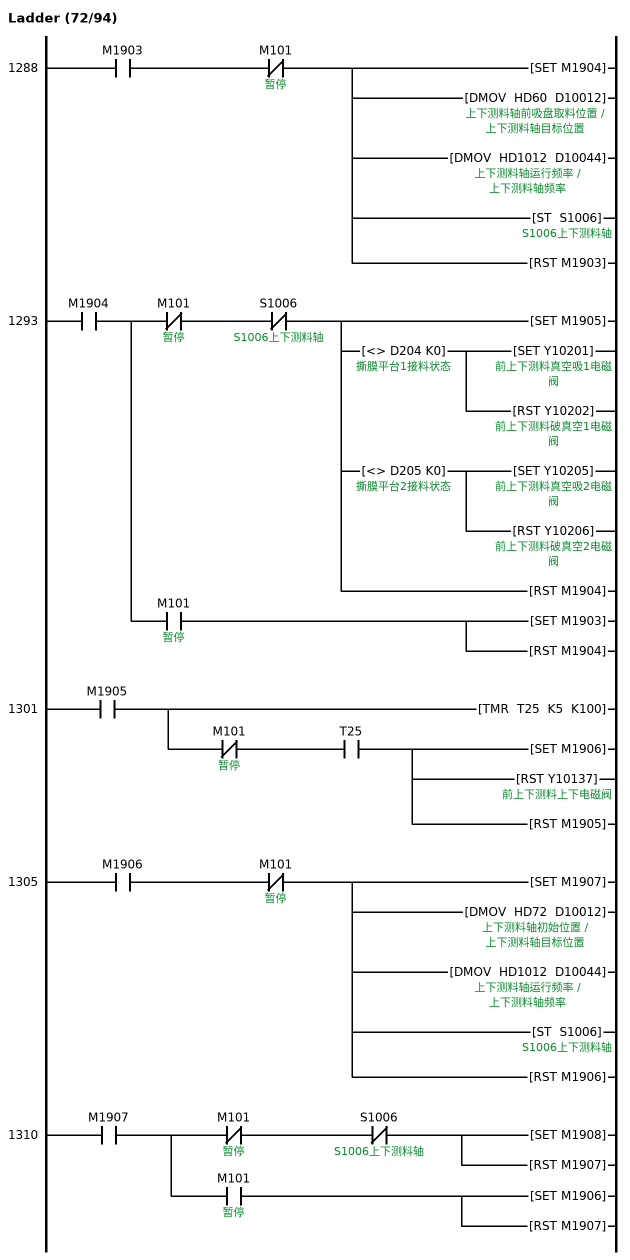
[picture p72: Ladder rows 1288-1310]
LD     M1903
ANI    M101	; 暂停
SET    M1904
DMOV   HD60 D10012	; 上下测料轴前吸盘取料位置 / 上下测料轴目标位置
DMOV   HD1012 D10044	; 上下测料轴运行频率 / 上下测料轴频率
ST     S1006	; S1006上下测料轴
RST    M1903
LD     M1904
MPS
ANI    M101	; 暂停
ANI    S1006	; S1006上下测料轴
SET    M1905
MPS
AND<>  D204 K0	; 撕膜平台1接料状态
SET    Y10201	; 前上下测料真空吸1电磁阀
RST    Y10202	; 前上下测料破真空1电磁阀
MRD
AND<>  D205 K0	; 撕膜平台2接料状态
SET    Y10205	; 前上下测料真空吸2电磁阀
RST    Y10206	; 前上下测料破真空2电磁阀
MPP
RST    M1904
MPP
AND    M101	; 暂停
SET    M1903
RST    M1904
LD     M1905
TMR    T25 K5 K100
ANI    M101	; 暂停
AND    T25
SET    M1906
RST    Y10137	; 前上下测料上下电磁阀
RST    M1905
LD     M1906
ANI    M101	; 暂停
SET    M1907
DMOV   HD72 D10012	; 上下测料轴初始位置 / 上下测料轴目标位置
DMOV   HD1012 D10044	; 上下测料轴运行频率 / 上下测料轴频率
ST     S1006	; S1006上下测料轴
RST    M1906
LD     M1907
MPS
ANI    M101	; 暂停
ANI    S1006	; S1006上下测料轴
SET    M1908
RST    M1907
MPP
AND    M101	; 暂停
SET    M1906
RST    M1907

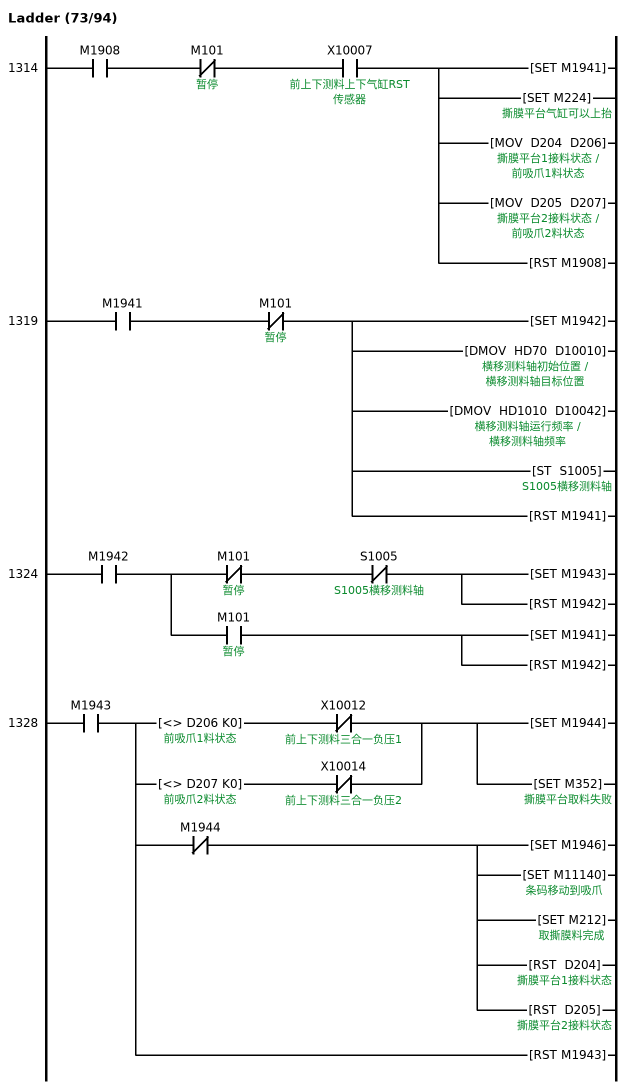
LD     M1908
ANI    M101	; 暂停
AND    X10007	; 前上下测料上下气缸RST传感器
SET    M1941
SET    M224	; 撕膜平台气缸可以上抬
MOV    D204 D206	; 撕膜平台1接料状态 / 前吸爪1料状态
MOV    D205 D207	; 撕膜平台2接料状态 / 前吸爪2料状态
RST    M1908
LD     M1941
ANI    M101	; 暂停
SET    M1942
DMOV   HD70 D10010	; 横移测料轴初始位置 / 横移测料轴目标位置
DMOV   HD1010 D10042	; 横移测料轴运行频率 / 横移测料轴频率
ST     S1005	; S1005横移测料轴
RST    M1941
LD     M1942
MPS
ANI    M101	; 暂停
ANI    S1005	; S1005横移测料轴
SET    M1943
RST    M1942
MPP
AND    M101	; 暂停
SET    M1941
RST    M1942
LD     M1943
MPS
LD<>   D206 K0	; 前吸爪1料状态
ANI    X10012	; 前上下测料三合一负压1
LD<>   D207 K0	; 前吸爪2料状态
ANI    X10014	; 前上下测料三合一负压2
ORB
ANB
SET    M1944
SET    M352	; 撕膜平台取料失败
MRD
ANI    M1944
SET    M1946
SET    M11140	; 条码移动到吸爪
SET    M212	; 取撕膜料完成
RST    D204	; 撕膜平台1接料状态
RST    D205	; 撕膜平台2接料状态
MPP
RST    M1943

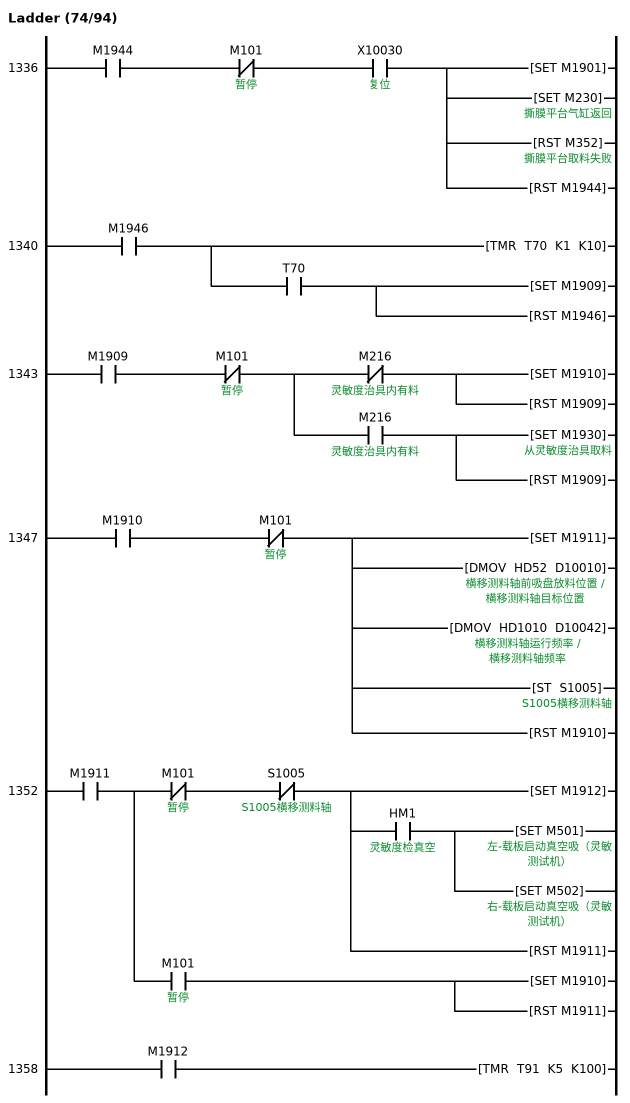
LD     M1944
ANI    M101	; 暂停
AND    X10030	; 复位
SET    M1901
SET    M230	; 撕膜平台气缸返回
RST    M352	; 撕膜平台取料失败
RST    M1944
LD     M1946
TMR    T70 K1 K10
AND    T70
SET    M1909
RST    M1946
LD     M1909
ANI    M101	; 暂停
MPS
ANI    M216	; 灵敏度治具内有料
SET    M1910
RST    M1909
MPP
AND    M216	; 灵敏度治具内有料
SET    M1930	; 从灵敏度治具取料
RST    M1909
LD     M1910
ANI    M101	; 暂停
SET    M1911
DMOV   HD52 D10010	; 横移测料轴前吸盘放料位置 / 横移测料轴目标位置
DMOV   HD1010 D10042	; 横移测料轴运行频率 / 横移测料轴频率
ST     S1005	; S1005横移测料轴
RST    M1910
LD     M1911
MPS
ANI    M101	; 暂停
ANI    S1005	; S1005横移测料轴
SET    M1912
MPS
AND    HM1	; 灵敏度检真空
SET    M501	; 左-载板启动真空吸（灵敏测试机）
SET    M502	; 右-载板启动真空吸（灵敏测试机）
MPP
RST    M1911
MPP
AND    M101	; 暂停
SET    M1910
RST    M1911
LD     M1912
TMR    T91 K5 K100

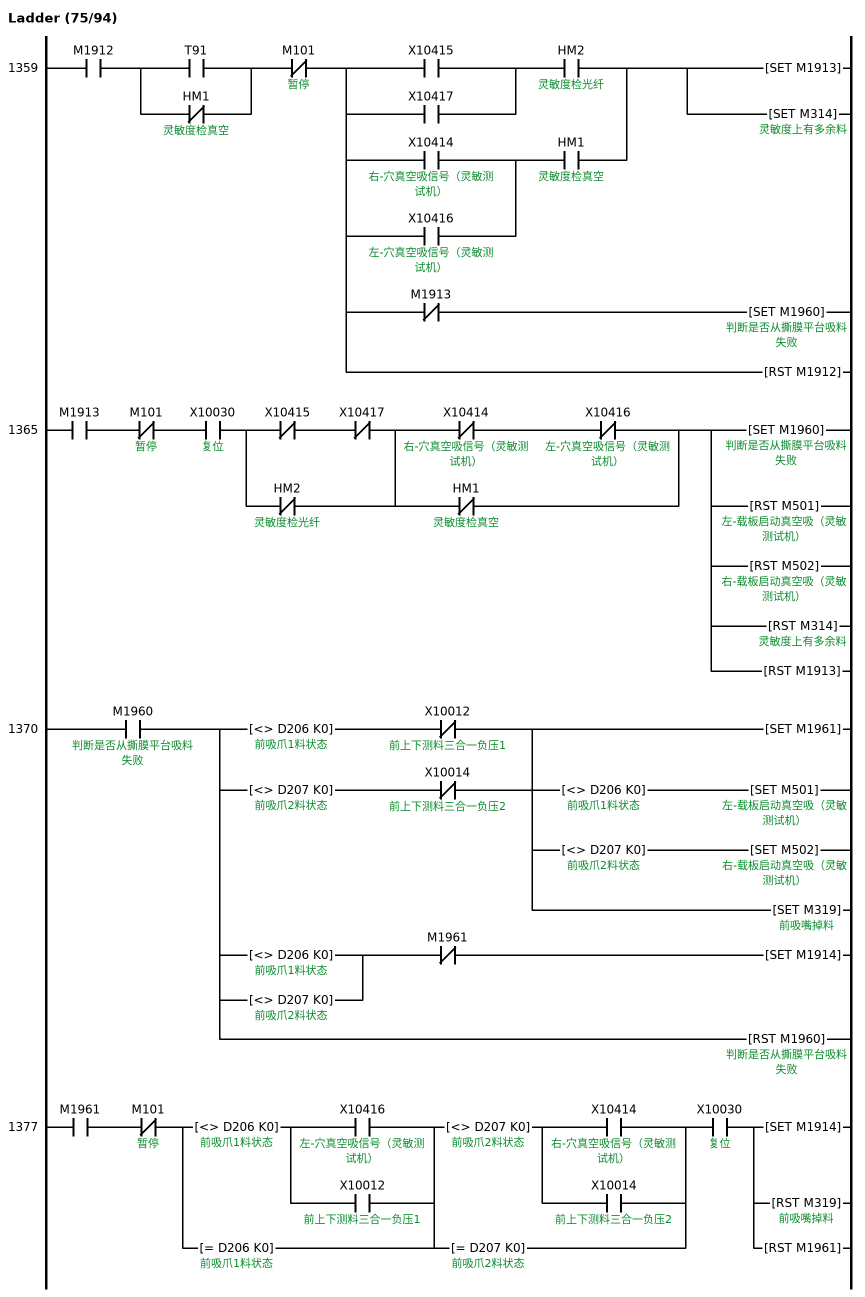
LD     M1912
LD     T91
ORI    HM1	; 灵敏度检真空
ANB
ANI    M101	; 暂停
MPS
LD     X10415
OR     X10417
AND    HM2	; 灵敏度检光纤
LD     X10414	; 右-穴真空吸信号（灵敏测试机）
OR     X10416	; 左-穴真空吸信号（灵敏测试机）
AND    HM1	; 灵敏度检真空
ORB
ANB
SET    M1913
SET    M314	; 灵敏度上有多余料
MRD
ANI    M1913
SET    M1960	; 判断是否从撕膜平台吸料失败
MPP
RST    M1912
LD     M1913
ANI    M101	; 暂停
AND    X10030	; 复位
LDI    X10415
ANI    X10417
ORI    HM2	; 灵敏度检光纤
ANB
LDI    X10414	; 右-穴真空吸信号（灵敏测试机）
ANI    X10416	; 左-穴真空吸信号（灵敏测试机）
ORI    HM1	; 灵敏度检真空
ANB
SET    M1960	; 判断是否从撕膜平台吸料失败
RST    M501	; 左-载板启动真空吸（灵敏测试机）
RST    M502	; 右-载板启动真空吸（灵敏测试机）
RST    M314	; 灵敏度上有多余料
RST    M1913
LD     M1960	; 判断是否从撕膜平台吸料失败
MPS
LD<>   D206 K0	; 前吸爪1料状态
ANI    X10012	; 前上下测料三合一负压1
LD<>   D207 K0	; 前吸爪2料状态
ANI    X10014	; 前上下测料三合一负压2
ORB
ANB
SET    M1961
MPS
AND<>  D206 K0	; 前吸爪1料状态
SET    M501	; 左-载板启动真空吸（灵敏测试机）
MRD
AND<>  D207 K0	; 前吸爪2料状态
SET    M502	; 右-载板启动真空吸（灵敏测试机）
MPP
SET    M319	; 前吸嘴掉料
MRD
LD<>   D206 K0	; 前吸爪1料状态
OR<>   D207 K0	; 前吸爪2料状态
ANB
ANI    M1961
SET    M1914
MPP
RST    M1960	; 判断是否从撕膜平台吸料失败
LD     M1961
ANI    M101	; 暂停
LD<>   D206 K0	; 前吸爪1料状态
LD     X10416	; 左-穴真空吸信号（灵敏测试机）
OR     X10012	; 前上下测料三合一负压1
ANB
OR=    D206 K0	; 前吸爪1料状态
ANB
LD<>   D207 K0	; 前吸爪2料状态
LD     X10414	; 右-穴真空吸信号（灵敏测试机）
OR     X10014	; 前上下测料三合一负压2
ANB
OR=    D207 K0	; 前吸爪2料状态
ANB
AND    X10030	; 复位
SET    M1914
RST    M319	; 前吸嘴掉料
RST    M1961

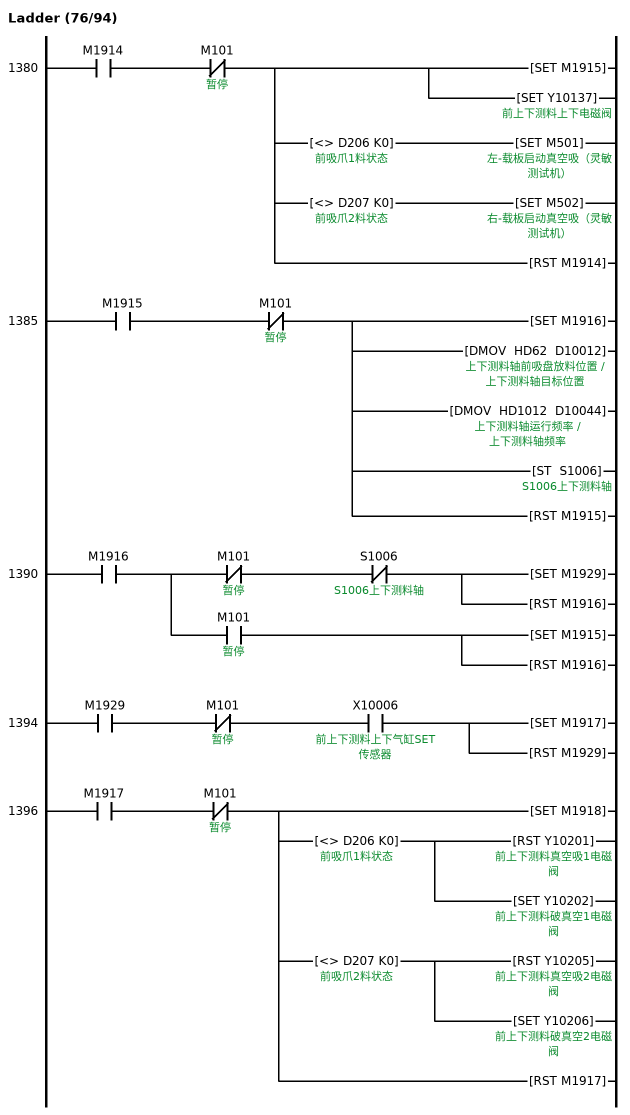
LD     M1914
ANI    M101	; 暂停
SET    M1915
SET    Y10137	; 前上下测料上下电磁阀
MPS
AND<>  D206 K0	; 前吸爪1料状态
SET    M501	; 左-载板启动真空吸（灵敏测试机）
MRD
AND<>  D207 K0	; 前吸爪2料状态
SET    M502	; 右-载板启动真空吸（灵敏测试机）
MPP
RST    M1914
LD     M1915
ANI    M101	; 暂停
SET    M1916
DMOV   HD62 D10012	; 上下测料轴前吸盘放料位置 / 上下测料轴目标位置
DMOV   HD1012 D10044	; 上下测料轴运行频率 / 上下测料轴频率
ST     S1006	; S1006上下测料轴
RST    M1915
LD     M1916
MPS
ANI    M101	; 暂停
ANI    S1006	; S1006上下测料轴
SET    M1929
RST    M1916
MPP
AND    M101	; 暂停
SET    M1915
RST    M1916
LD     M1929
ANI    M101	; 暂停
AND    X10006	; 前上下测料上下气缸SET传感器
SET    M1917
RST    M1929
LD     M1917
ANI    M101	; 暂停
SET    M1918
MPS
AND<>  D206 K0	; 前吸爪1料状态
RST    Y10201	; 前上下测料真空吸1电磁阀
SET    Y10202	; 前上下测料破真空1电磁阀
MRD
AND<>  D207 K0	; 前吸爪2料状态
RST    Y10205	; 前上下测料真空吸2电磁阀
SET    Y10206	; 前上下测料破真空2电磁阀
MPP
RST    M1917

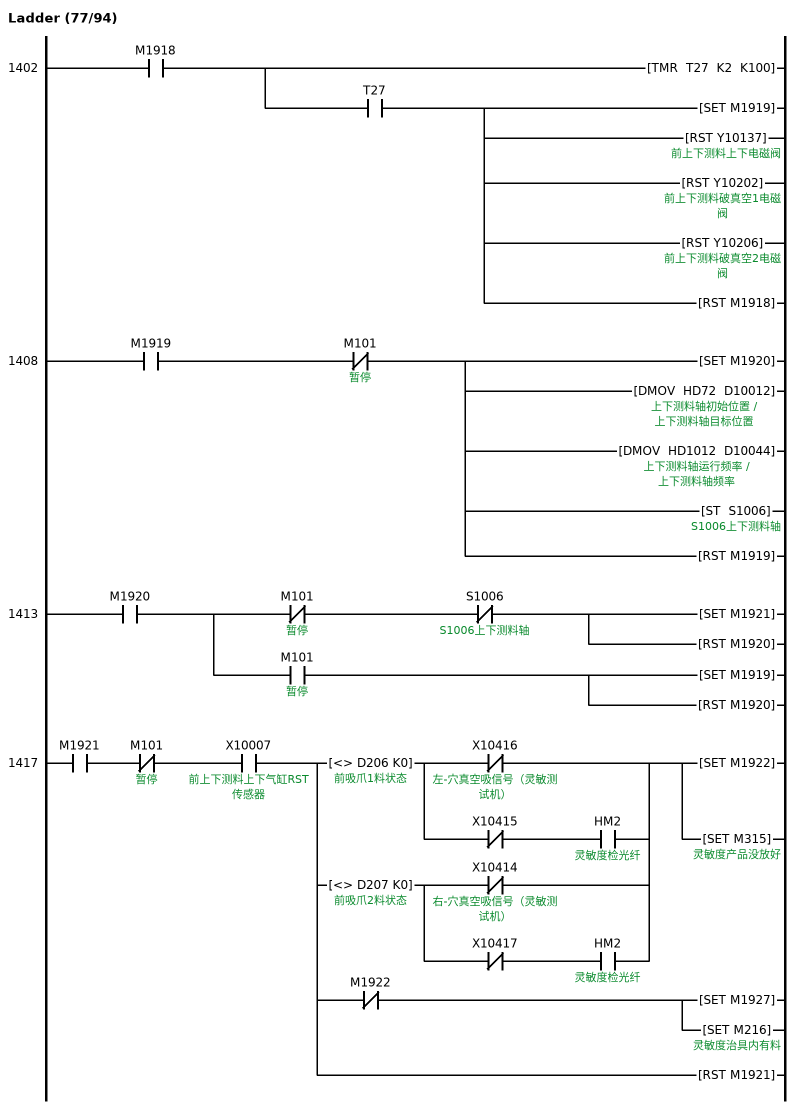
LD     M1918
TMR    T27 K2 K100
AND    T27
SET    M1919
RST    Y10137	; 前上下测料上下电磁阀
RST    Y10202	; 前上下测料破真空1电磁阀
RST    Y10206	; 前上下测料破真空2电磁阀
RST    M1918
LD     M1919
ANI    M101	; 暂停
SET    M1920
DMOV   HD72 D10012	; 上下测料轴初始位置 / 上下测料轴目标位置
DMOV   HD1012 D10044	; 上下测料轴运行频率 / 上下测料轴频率
ST     S1006	; S1006上下测料轴
RST    M1919
LD     M1920
MPS
ANI    M101	; 暂停
ANI    S1006	; S1006上下测料轴
SET    M1921
RST    M1920
MPP
AND    M101	; 暂停
SET    M1919
RST    M1920
LD     M1921
ANI    M101	; 暂停
AND    X10007	; 前上下测料上下气缸RST传感器
MPS
LD<>   D206 K0	; 前吸爪1料状态
LDI    X10416	; 左-穴真空吸信号（灵敏测试机）
LDI    X10415
AND    HM2	; 灵敏度检光纤
ORB
ANB
LD<>   D207 K0	; 前吸爪2料状态
LDI    X10414	; 右-穴真空吸信号（灵敏测试机）
LDI    X10417
AND    HM2	; 灵敏度检光纤
ORB
ANB
ORB
ANB
SET    M1922
SET    M315	; 灵敏度产品没放好
MRD
ANI    M1922
SET    M1927
SET    M216	; 灵敏度治具内有料
MPP
RST    M1921

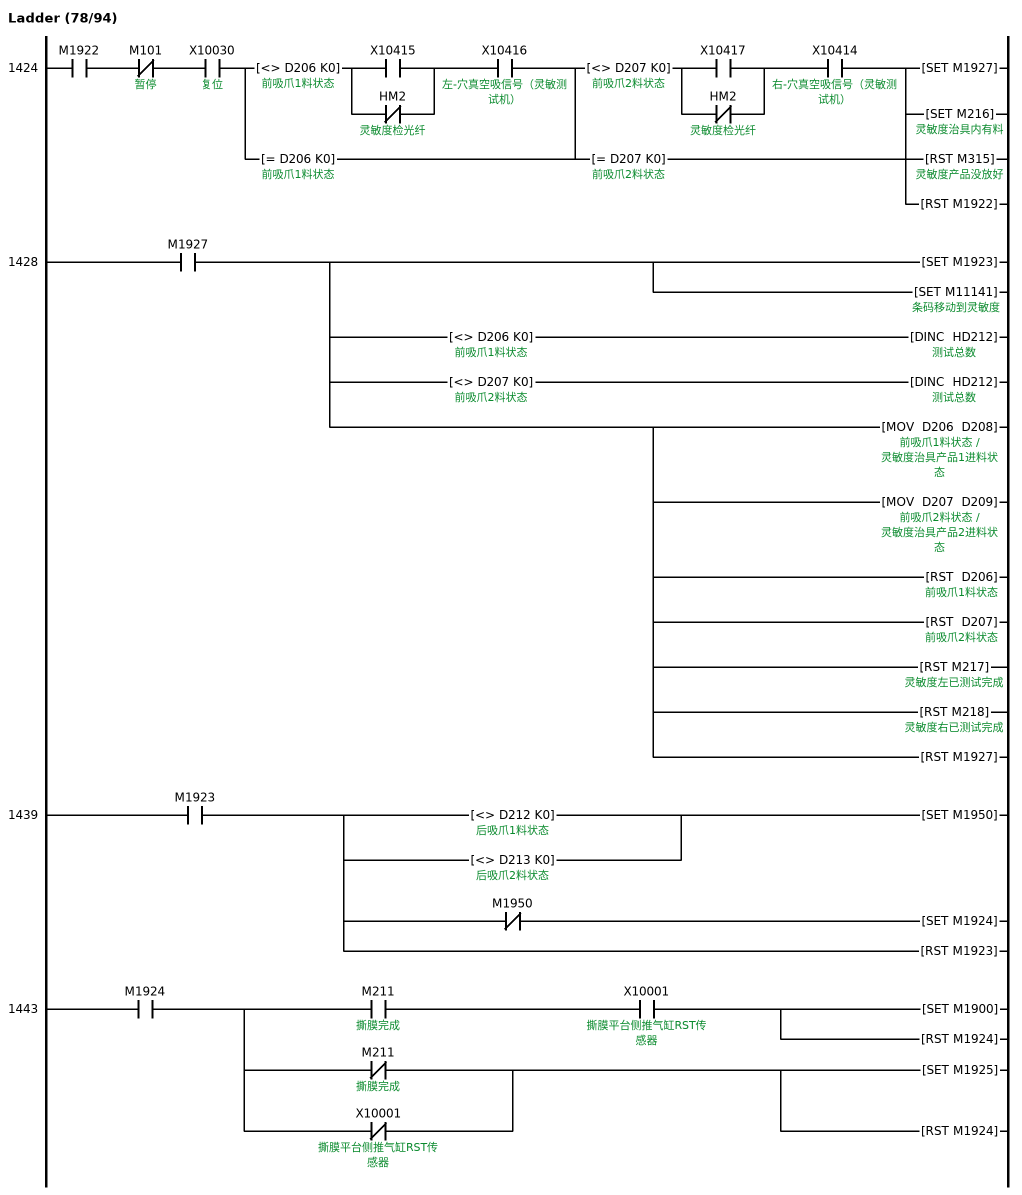
LD     M1922
ANI    M101	; 暂停
AND    X10030	; 复位
LD<>   D206 K0	; 前吸爪1料状态
LD     X10415
ORI    HM2	; 灵敏度检光纤
ANB
AND    X10416	; 左-穴真空吸信号（灵敏测试机）
OR=    D206 K0	; 前吸爪1料状态
ANB
LD<>   D207 K0	; 前吸爪2料状态
LD     X10417
ORI    HM2	; 灵敏度检光纤
ANB
AND    X10414	; 右-穴真空吸信号（灵敏测试机）
OR=    D207 K0	; 前吸爪2料状态
ANB
SET    M1927
SET    M216	; 灵敏度治具内有料
RST    M315	; 灵敏度产品没放好
RST    M1922
LD     M1927
SET    M1923
SET    M11141	; 条码移动到灵敏度
MPS
AND<>  D206 K0	; 前吸爪1料状态
DINC   HD212	; 测试总数
MRD
AND<>  D207 K0	; 前吸爪2料状态
DINC   HD212	; 测试总数
MPP
MOV    D206 D208	; 前吸爪1料状态 / 灵敏度治具产品1进料状态
MOV    D207 D209	; 前吸爪2料状态 / 灵敏度治具产品2进料状态
RST    D206	; 前吸爪1料状态
RST    D207	; 前吸爪2料状态
RST    M217	; 灵敏度左已测试完成
RST    M218	; 灵敏度右已测试完成
RST    M1927
LD     M1923
MPS
LD<>   D212 K0	; 后吸爪1料状态
OR<>   D213 K0	; 后吸爪2料状态
ANB
SET    M1950
MRD
ANI    M1950
SET    M1924
MPP
RST    M1923
LD     M1924
MPS
AND    M211	; 撕膜完成
AND    X10001	; 撕膜平台侧推气缸RST传感器
SET    M1900
RST    M1924
MPP
LDI    M211	; 撕膜完成
ORI    X10001	; 撕膜平台侧推气缸RST传感器
ANB
SET    M1925
RST    M1924

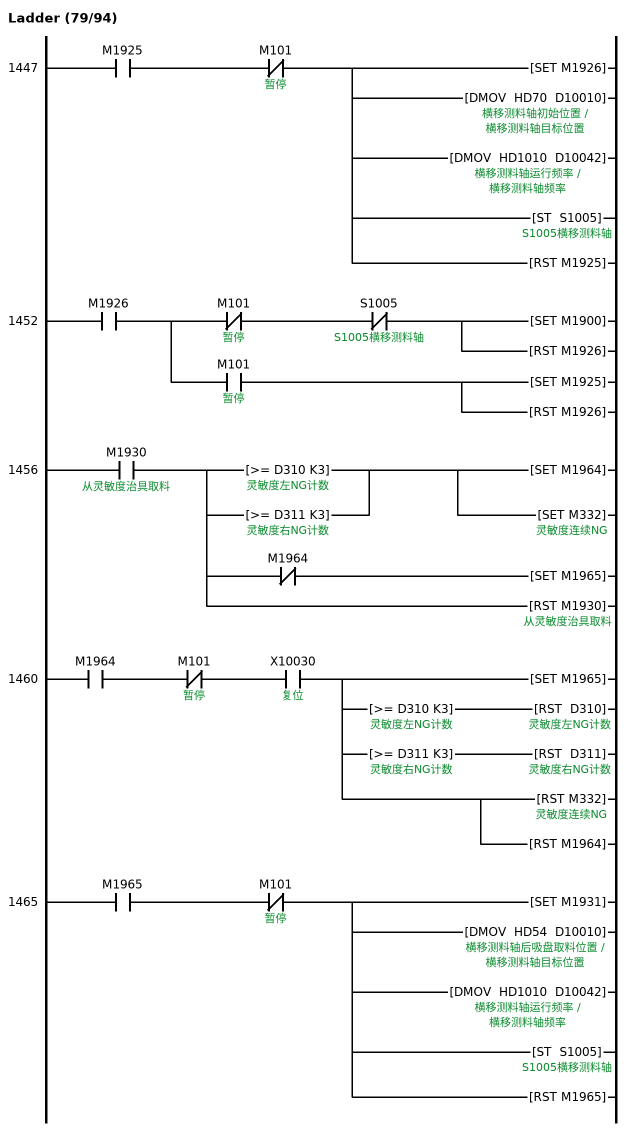
LD     M1925
ANI    M101	; 暂停
SET    M1926
DMOV   HD70 D10010	; 横移测料轴初始位置 / 横移测料轴目标位置
DMOV   HD1010 D10042	; 横移测料轴运行频率 / 横移测料轴频率
ST     S1005	; S1005横移测料轴
RST    M1925
LD     M1926
MPS
ANI    M101	; 暂停
ANI    S1005	; S1005横移测料轴
SET    M1900
RST    M1926
MPP
AND    M101	; 暂停
SET    M1925
RST    M1926
LD     M1930	; 从灵敏度治具取料
MPS
LD>=   D310 K3	; 灵敏度左NG计数
OR>=   D311 K3	; 灵敏度右NG计数
ANB
SET    M1964
SET    M332	; 灵敏度连续NG
MRD
ANI    M1964
SET    M1965
MPP
RST    M1930	; 从灵敏度治具取料
LD     M1964
ANI    M101	; 暂停
AND    X10030	; 复位
SET    M1965
MPS
AND>=  D310 K3	; 灵敏度左NG计数
RST    D310	; 灵敏度左NG计数
MRD
AND>=  D311 K3	; 灵敏度右NG计数
RST    D311	; 灵敏度右NG计数
MPP
RST    M332	; 灵敏度连续NG
RST    M1964
LD     M1965
ANI    M101	; 暂停
SET    M1931
DMOV   HD54 D10010	; 横移测料轴后吸盘取料位置 / 横移测料轴目标位置
DMOV   HD1010 D10042	; 横移测料轴运行频率 / 横移测料轴频率
ST     S1005	; S1005横移测料轴
RST    M1965

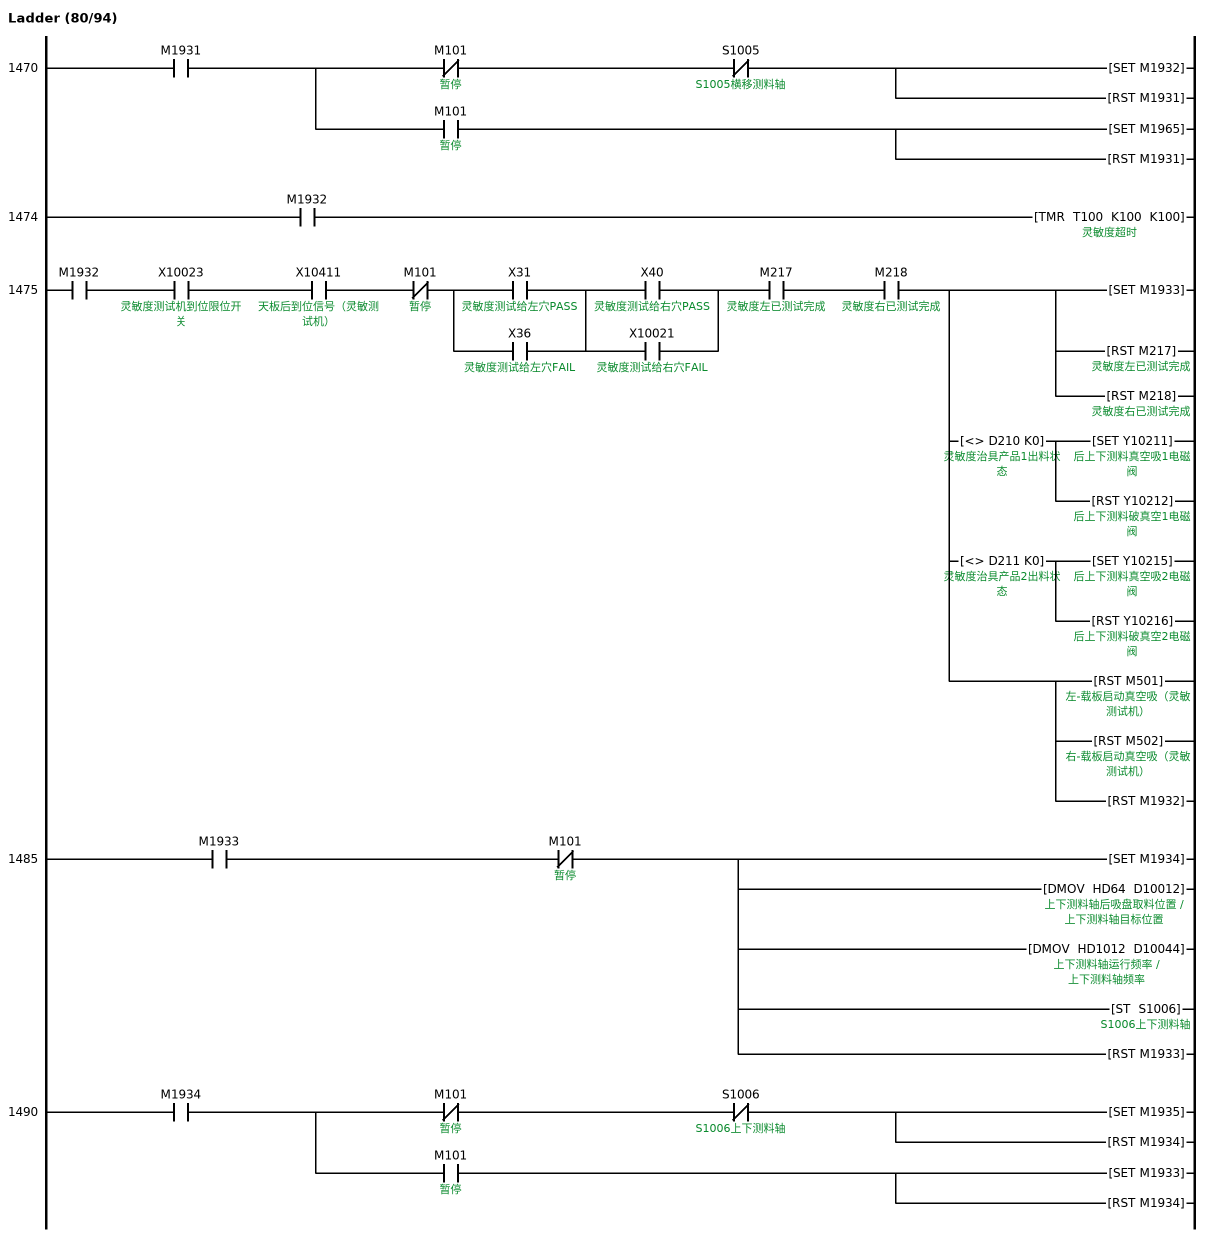
LD     M1931
MPS
ANI    M101	; 暂停
ANI    S1005	; S1005横移测料轴
SET    M1932
RST    M1931
MPP
AND    M101	; 暂停
SET    M1965
RST    M1931
LD     M1932
TMR    T100 K100 K100	; 灵敏度超时
LD     M1932
AND    X10023	; 灵敏度测试机到位限位开关
AND    X10411	; 天板后到位信号（灵敏测试机）
ANI    M101	; 暂停
LD     X31	; 灵敏度测试给左穴PASS
OR     X36	; 灵敏度测试给左穴FAIL
ANB
LD     X40	; 灵敏度测试给右穴PASS
OR     X10021	; 灵敏度测试给右穴FAIL
ANB
AND    M217	; 灵敏度左已测试完成
AND    M218	; 灵敏度右已测试完成
SET    M1933
RST    M217	; 灵敏度左已测试完成
RST    M218	; 灵敏度右已测试完成
MPS
AND<>  D210 K0	; 灵敏度治具产品1出料状态
SET    Y10211	; 后上下测料真空吸1电磁阀
RST    Y10212	; 后上下测料破真空1电磁阀
MRD
AND<>  D211 K0	; 灵敏度治具产品2出料状态
SET    Y10215	; 后上下测料真空吸2电磁阀
RST    Y10216	; 后上下测料破真空2电磁阀
MPP
RST    M501	; 左-载板启动真空吸（灵敏测试机）
RST    M502	; 右-载板启动真空吸（灵敏测试机）
RST    M1932
LD     M1933
ANI    M101	; 暂停
SET    M1934
DMOV   HD64 D10012	; 上下测料轴后吸盘取料位置 / 上下测料轴目标位置
DMOV   HD1012 D10044	; 上下测料轴运行频率 / 上下测料轴频率
ST     S1006	; S1006上下测料轴
RST    M1933
LD     M1934
MPS
ANI    M101	; 暂停
ANI    S1006	; S1006上下测料轴
SET    M1935
RST    M1934
MPP
AND    M101	; 暂停
SET    M1933
RST    M1934

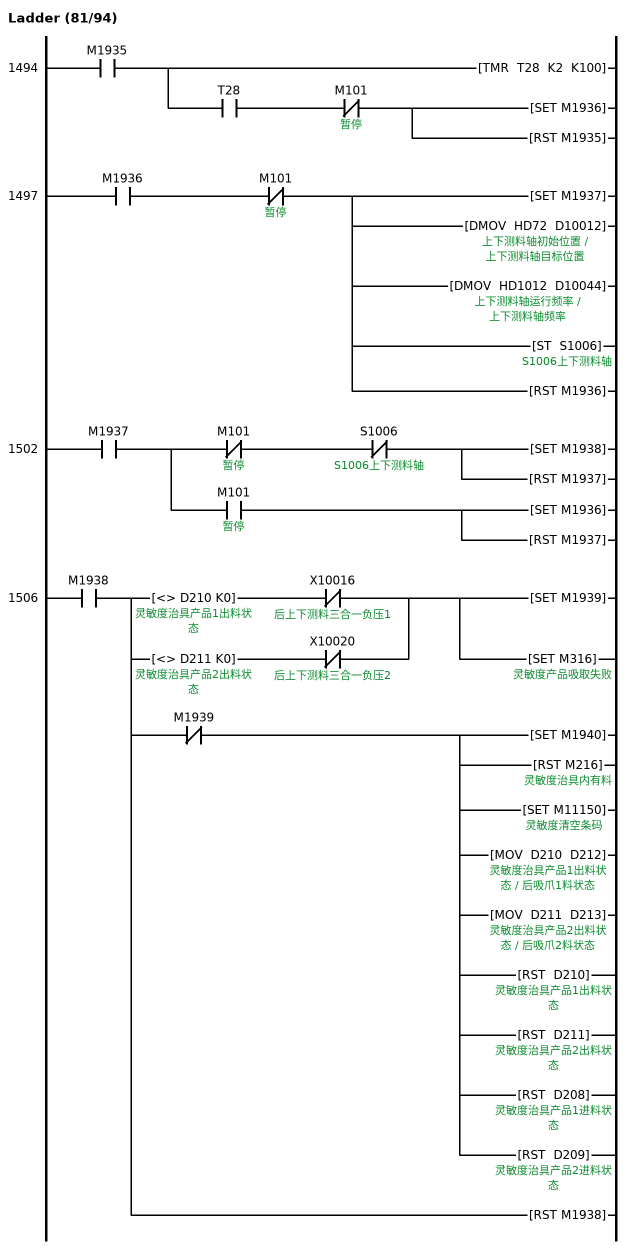
LD     M1935
TMR    T28 K2 K100
AND    T28
ANI    M101	; 暂停
SET    M1936
RST    M1935
LD     M1936
ANI    M101	; 暂停
SET    M1937
DMOV   HD72 D10012	; 上下测料轴初始位置 / 上下测料轴目标位置
DMOV   HD1012 D10044	; 上下测料轴运行频率 / 上下测料轴频率
ST     S1006	; S1006上下测料轴
RST    M1936
LD     M1937
MPS
ANI    M101	; 暂停
ANI    S1006	; S1006上下测料轴
SET    M1938
RST    M1937
MPP
AND    M101	; 暂停
SET    M1936
RST    M1937
LD     M1938
MPS
LD<>   D210 K0	; 灵敏度治具产品1出料状态
ANI    X10016	; 后上下测料三合一负压1
LD<>   D211 K0	; 灵敏度治具产品2出料状态
ANI    X10020	; 后上下测料三合一负压2
ORB
ANB
SET    M1939
SET    M316	; 灵敏度产品吸取失败
MRD
ANI    M1939
SET    M1940
RST    M216	; 灵敏度治具内有料
SET    M11150	; 灵敏度清空条码
MOV    D210 D212	; 灵敏度治具产品1出料状态 / 后吸爪1料状态
MOV    D211 D213	; 灵敏度治具产品2出料状态 / 后吸爪2料状态
RST    D210	; 灵敏度治具产品1出料状态
RST    D211	; 灵敏度治具产品2出料状态
RST    D208	; 灵敏度治具产品1进料状态
RST    D209	; 灵敏度治具产品2进料状态
MPP
RST    M1938

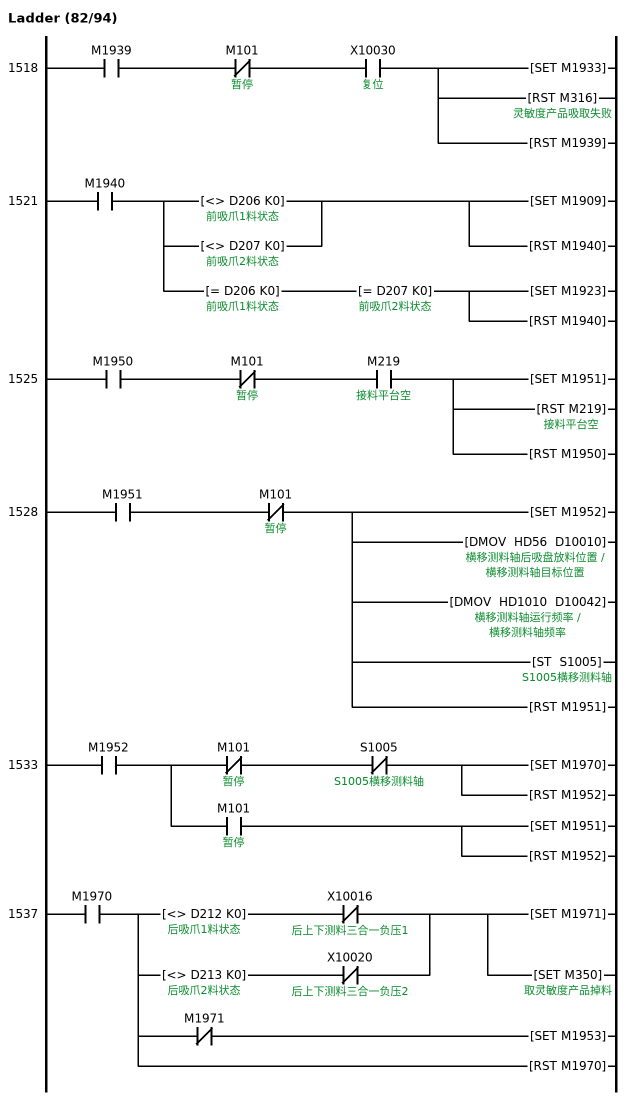
LD     M1939
ANI    M101	; 暂停
AND    X10030	; 复位
SET    M1933
RST    M316	; 灵敏度产品吸取失败
RST    M1939
LD     M1940
MPS
LD<>   D206 K0	; 前吸爪1料状态
OR<>   D207 K0	; 前吸爪2料状态
ANB
SET    M1909
RST    M1940
MPP
AND=   D206 K0	; 前吸爪1料状态
AND=   D207 K0	; 前吸爪2料状态
SET    M1923
RST    M1940
LD     M1950
ANI    M101	; 暂停
AND    M219	; 接料平台空
SET    M1951
RST    M219	; 接料平台空
RST    M1950
LD     M1951
ANI    M101	; 暂停
SET    M1952
DMOV   HD56 D10010	; 横移测料轴后吸盘放料位置 / 横移测料轴目标位置
DMOV   HD1010 D10042	; 横移测料轴运行频率 / 横移测料轴频率
ST     S1005	; S1005横移测料轴
RST    M1951
LD     M1952
MPS
ANI    M101	; 暂停
ANI    S1005	; S1005横移测料轴
SET    M1970
RST    M1952
MPP
AND    M101	; 暂停
SET    M1951
RST    M1952
LD     M1970
MPS
LD<>   D212 K0	; 后吸爪1料状态
ANI    X10016	; 后上下测料三合一负压1
LD<>   D213 K0	; 后吸爪2料状态
ANI    X10020	; 后上下测料三合一负压2
ORB
ANB
SET    M1971
SET    M350	; 取灵敏度产品掉料
MRD
ANI    M1971
SET    M1953
MPP
RST    M1970

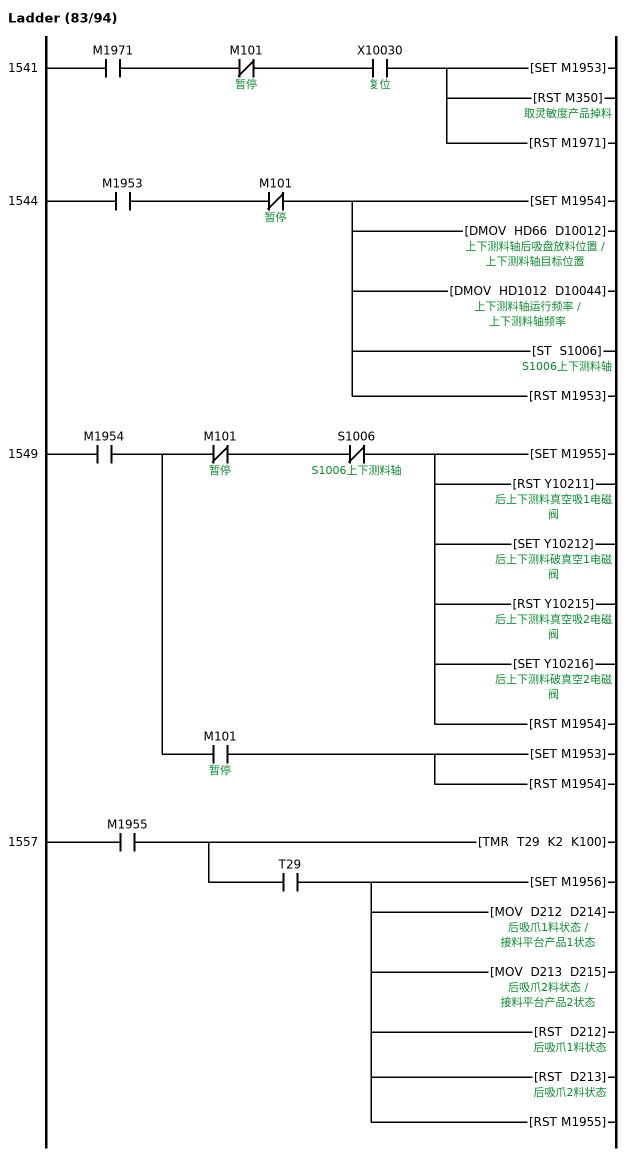
LD     M1971
ANI    M101	; 暂停
AND    X10030	; 复位
SET    M1953
RST    M350	; 取灵敏度产品掉料
RST    M1971
LD     M1953
ANI    M101	; 暂停
SET    M1954
DMOV   HD66 D10012	; 上下测料轴后吸盘放料位置 / 上下测料轴目标位置
DMOV   HD1012 D10044	; 上下测料轴运行频率 / 上下测料轴频率
ST     S1006	; S1006上下测料轴
RST    M1953
LD     M1954
MPS
ANI    M101	; 暂停
ANI    S1006	; S1006上下测料轴
SET    M1955
RST    Y10211	; 后上下测料真空吸1电磁阀
SET    Y10212	; 后上下测料破真空1电磁阀
RST    Y10215	; 后上下测料真空吸2电磁阀
SET    Y10216	; 后上下测料破真空2电磁阀
RST    M1954
MPP
AND    M101	; 暂停
SET    M1953
RST    M1954
LD     M1955
TMR    T29 K2 K100
AND    T29
SET    M1956
MOV    D212 D214	; 后吸爪1料状态 / 接料平台产品1状态
MOV    D213 D215	; 后吸爪2料状态 / 接料平台产品2状态
RST    D212	; 后吸爪1料状态
RST    D213	; 后吸爪2料状态
RST    M1955

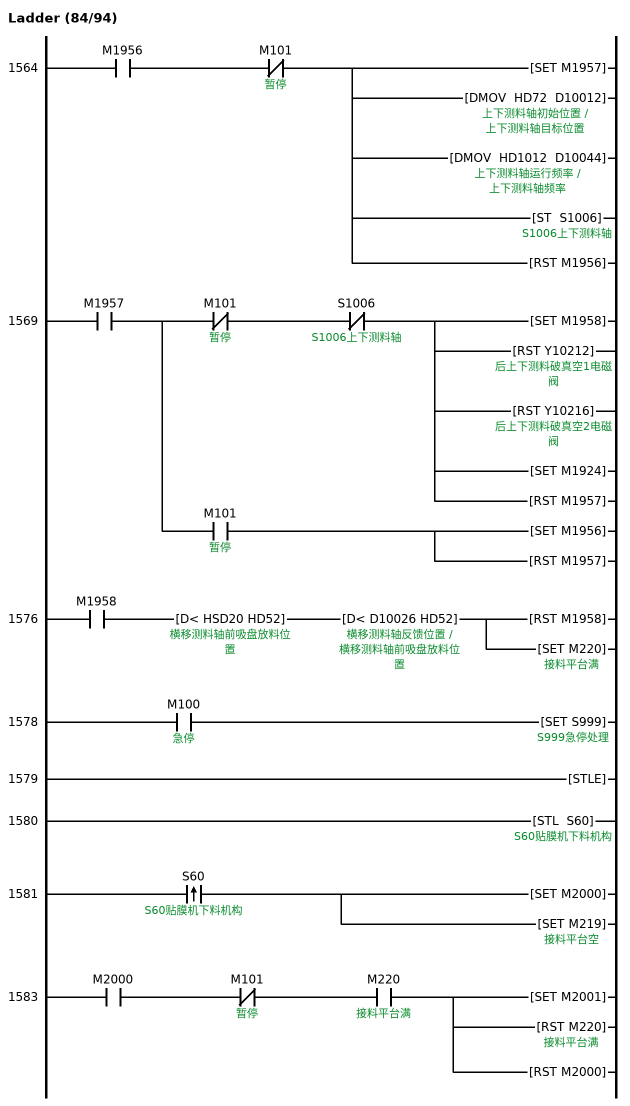
LD     M1956
ANI    M101	; 暂停
SET    M1957
DMOV   HD72 D10012	; 上下测料轴初始位置 / 上下测料轴目标位置
DMOV   HD1012 D10044	; 上下测料轴运行频率 / 上下测料轴频率
ST     S1006	; S1006上下测料轴
RST    M1956
LD     M1957
MPS
ANI    M101	; 暂停
ANI    S1006	; S1006上下测料轴
SET    M1958
RST    Y10212	; 后上下测料破真空1电磁阀
RST    Y10216	; 后上下测料破真空2电磁阀
SET    M1924
RST    M1957
MPP
AND    M101	; 暂停
SET    M1956
RST    M1957
LD     M1958
DAND<  HSD20 HD52	; 横移测料轴前吸盘放料位置
DAND<  D10026 HD52	; 横移测料轴反馈位置 / 横移测料轴前吸盘放料位置
RST    M1958
SET    M220	; 接料平台满
LD     M100	; 急停
SET    S999	; S999急停处理
STLE
STL    S60	; S60贴膜机下料机构
LDP    S60	; S60贴膜机下料机构
SET    M2000
SET    M219	; 接料平台空
LD     M2000
ANI    M101	; 暂停
AND    M220	; 接料平台满
SET    M2001
RST    M220	; 接料平台满
RST    M2000

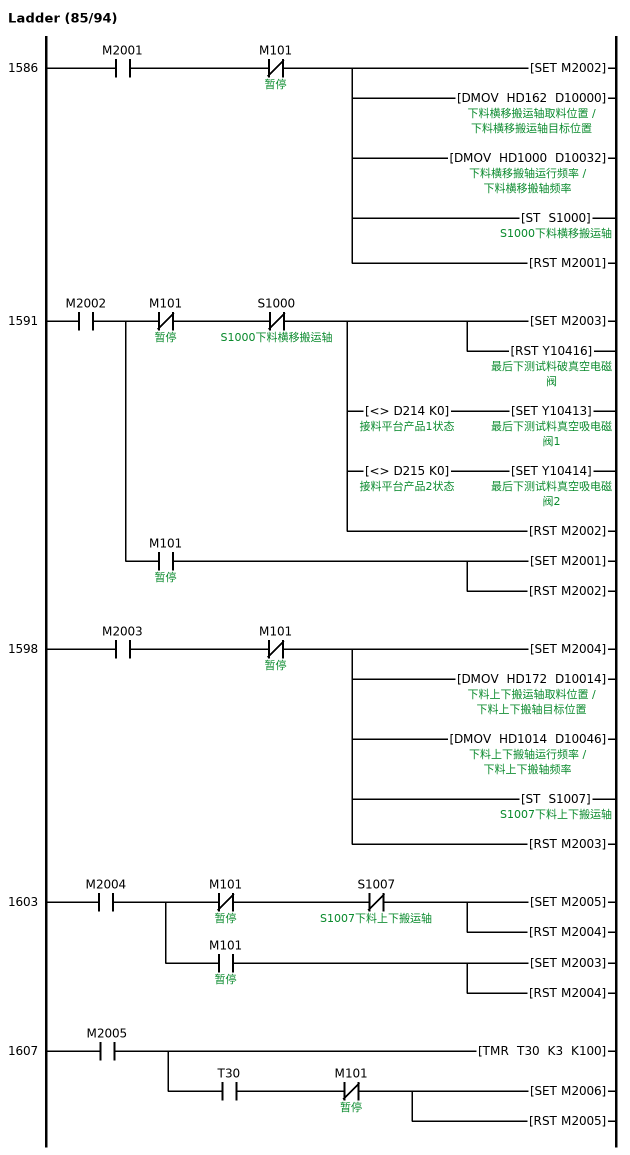
LD     M2001
ANI    M101	; 暂停
SET    M2002
DMOV   HD162 D10000	; 下料横移搬运轴取料位置 / 下料横移搬运轴目标位置
DMOV   HD1000 D10032	; 下料横移搬轴运行频率 / 下料横移搬轴频率
ST     S1000	; S1000下料横移搬运轴
RST    M2001
LD     M2002
MPS
ANI    M101	; 暂停
ANI    S1000	; S1000下料横移搬运轴
SET    M2003
RST    Y10416	; 最后下测试料破真空电磁阀
MPS
AND<>  D214 K0	; 接料平台产品1状态
SET    Y10413	; 最后下测试料真空吸电磁阀1
MRD
AND<>  D215 K0	; 接料平台产品2状态
SET    Y10414	; 最后下测试料真空吸电磁阀2
MPP
RST    M2002
MPP
AND    M101	; 暂停
SET    M2001
RST    M2002
LD     M2003
ANI    M101	; 暂停
SET    M2004
DMOV   HD172 D10014	; 下料上下搬运轴取料位置 / 下料上下搬轴目标位置
DMOV   HD1014 D10046	; 下料上下搬轴运行频率 / 下料上下搬轴频率
ST     S1007	; S1007下料上下搬运轴
RST    M2003
LD     M2004
MPS
ANI    M101	; 暂停
ANI    S1007	; S1007下料上下搬运轴
SET    M2005
RST    M2004
MPP
AND    M101	; 暂停
SET    M2003
RST    M2004
LD     M2005
TMR    T30 K3 K100
AND    T30
ANI    M101	; 暂停
SET    M2006
RST    M2005

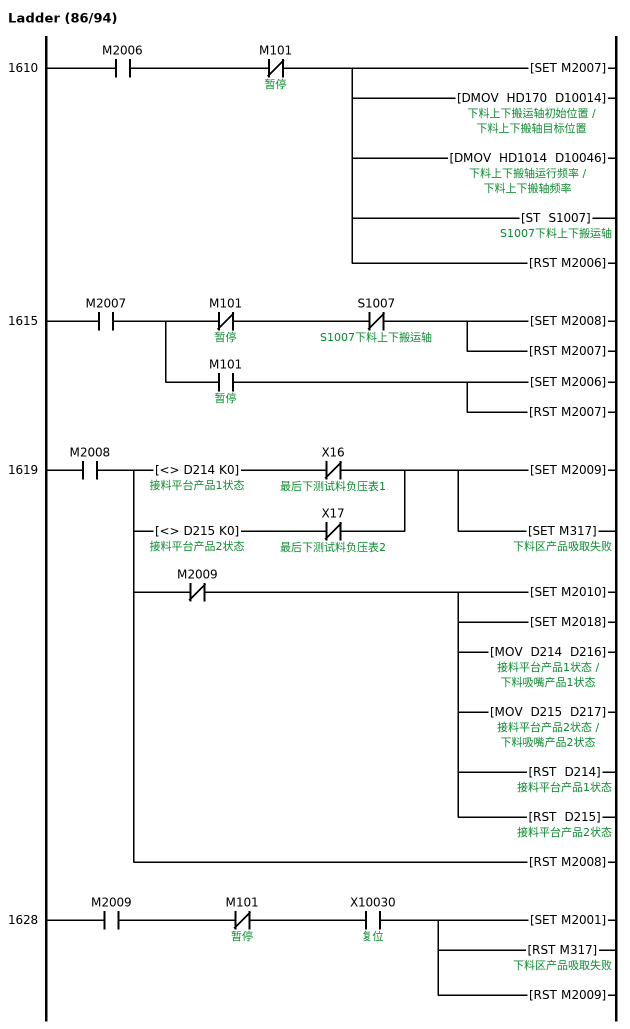
LD     M2006
ANI    M101	; 暂停
SET    M2007
DMOV   HD170 D10014	; 下料上下搬运轴初始位置 / 下料上下搬轴目标位置
DMOV   HD1014 D10046	; 下料上下搬轴运行频率 / 下料上下搬轴频率
ST     S1007	; S1007下料上下搬运轴
RST    M2006
LD     M2007
MPS
ANI    M101	; 暂停
ANI    S1007	; S1007下料上下搬运轴
SET    M2008
RST    M2007
MPP
AND    M101	; 暂停
SET    M2006
RST    M2007
LD     M2008
MPS
LD<>   D214 K0	; 接料平台产品1状态
ANI    X16	; 最后下测试料负压表1
LD<>   D215 K0	; 接料平台产品2状态
ANI    X17	; 最后下测试料负压表2
ORB
ANB
SET    M2009
SET    M317	; 下料区产品吸取失败
MRD
ANI    M2009
SET    M2010
SET    M2018
MOV    D214 D216	; 接料平台产品1状态 / 下料吸嘴产品1状态
MOV    D215 D217	; 接料平台产品2状态 / 下料吸嘴产品2状态
RST    D214	; 接料平台产品1状态
RST    D215	; 接料平台产品2状态
MPP
RST    M2008
LD     M2009
ANI    M101	; 暂停
AND    X10030	; 复位
SET    M2001
RST    M317	; 下料区产品吸取失败
RST    M2009

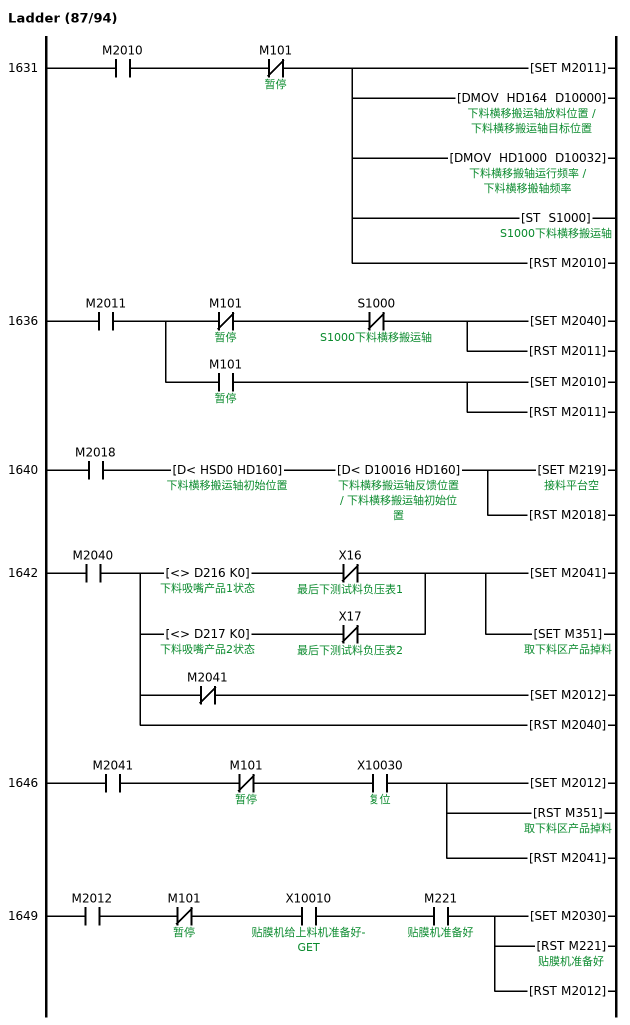
LD     M2010
ANI    M101	; 暂停
SET    M2011
DMOV   HD164 D10000	; 下料横移搬运轴放料位置 / 下料横移搬运轴目标位置
DMOV   HD1000 D10032	; 下料横移搬轴运行频率 / 下料横移搬轴频率
ST     S1000	; S1000下料横移搬运轴
RST    M2010
LD     M2011
MPS
ANI    M101	; 暂停
ANI    S1000	; S1000下料横移搬运轴
SET    M2040
RST    M2011
MPP
AND    M101	; 暂停
SET    M2010
RST    M2011
LD     M2018
DAND<  HSD0 HD160	; 下料横移搬运轴初始位置
DAND<  D10016 HD160	; 下料横移搬运轴反馈位置 / 下料横移搬运轴初始位置
SET    M219	; 接料平台空
RST    M2018
LD     M2040
MPS
LD<>   D216 K0	; 下料吸嘴产品1状态
ANI    X16	; 最后下测试料负压表1
LD<>   D217 K0	; 下料吸嘴产品2状态
ANI    X17	; 最后下测试料负压表2
ORB
ANB
SET    M2041
SET    M351	; 取下料区产品掉料
MRD
ANI    M2041
SET    M2012
MPP
RST    M2040
LD     M2041
ANI    M101	; 暂停
AND    X10030	; 复位
SET    M2012
RST    M351	; 取下料区产品掉料
RST    M2041
LD     M2012
ANI    M101	; 暂停
AND    X10010	; 贴膜机给上料机准备好-GET
AND    M221	; 贴膜机准备好
SET    M2030
RST    M221	; 贴膜机准备好
RST    M2012

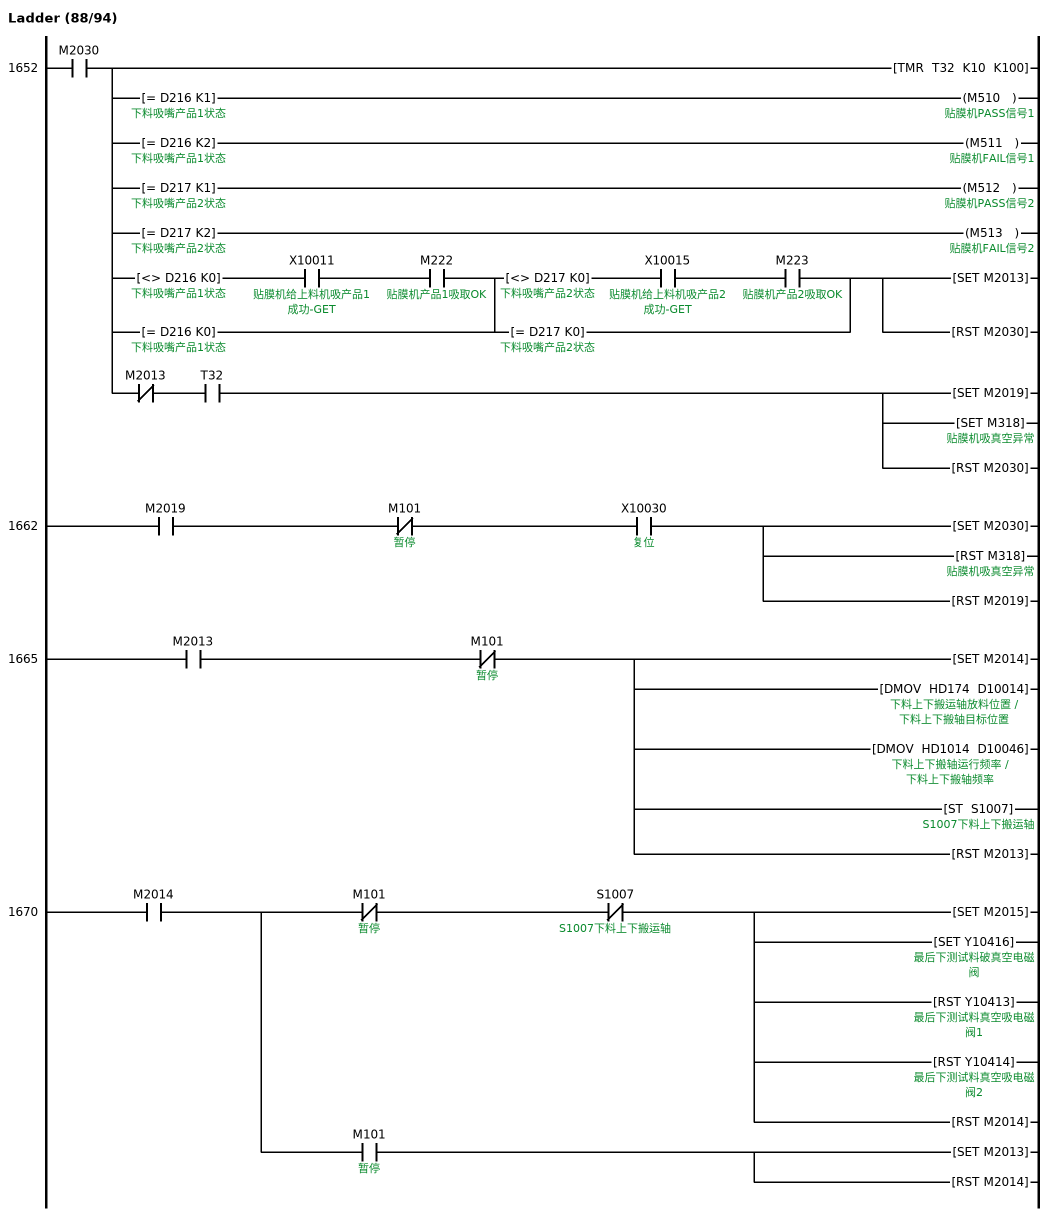
LD     M2030
TMR    T32 K10 K100
MPS
AND=   D216 K1	; 下料吸嘴产品1状态
OUT    M510	; 贴膜机PASS信号1
MRD
AND=   D216 K2	; 下料吸嘴产品1状态
OUT    M511	; 贴膜机FAIL信号1
MRD
AND=   D217 K1	; 下料吸嘴产品2状态
OUT    M512	; 贴膜机PASS信号2
MRD
AND=   D217 K2	; 下料吸嘴产品2状态
OUT    M513	; 贴膜机FAIL信号2
MRD
LD<>   D216 K0	; 下料吸嘴产品1状态
AND    X10011	; 贴膜机给上料机吸产品1成功-GET
AND    M222	; 贴膜机产品1吸取OK
OR=    D216 K0	; 下料吸嘴产品1状态
ANB
LD<>   D217 K0	; 下料吸嘴产品2状态
AND    X10015	; 贴膜机给上料机吸产品2成功-GET
AND    M223	; 贴膜机产品2吸取OK
OR=    D217 K0	; 下料吸嘴产品2状态
ANB
SET    M2013
RST    M2030
MPP
ANI    M2013
AND    T32
SET    M2019
SET    M318	; 贴膜机吸真空异常
RST    M2030
LD     M2019
ANI    M101	; 暂停
AND    X10030	; 复位
SET    M2030
RST    M318	; 贴膜机吸真空异常
RST    M2019
LD     M2013
ANI    M101	; 暂停
SET    M2014
DMOV   HD174 D10014	; 下料上下搬运轴放料位置 / 下料上下搬轴目标位置
DMOV   HD1014 D10046	; 下料上下搬轴运行频率 / 下料上下搬轴频率
ST     S1007	; S1007下料上下搬运轴
RST    M2013
LD     M2014
MPS
ANI    M101	; 暂停
ANI    S1007	; S1007下料上下搬运轴
SET    M2015
SET    Y10416	; 最后下测试料破真空电磁阀
RST    Y10413	; 最后下测试料真空吸电磁阀1
RST    Y10414	; 最后下测试料真空吸电磁阀2
RST    M2014
MPP
AND    M101	; 暂停
SET    M2013
RST    M2014

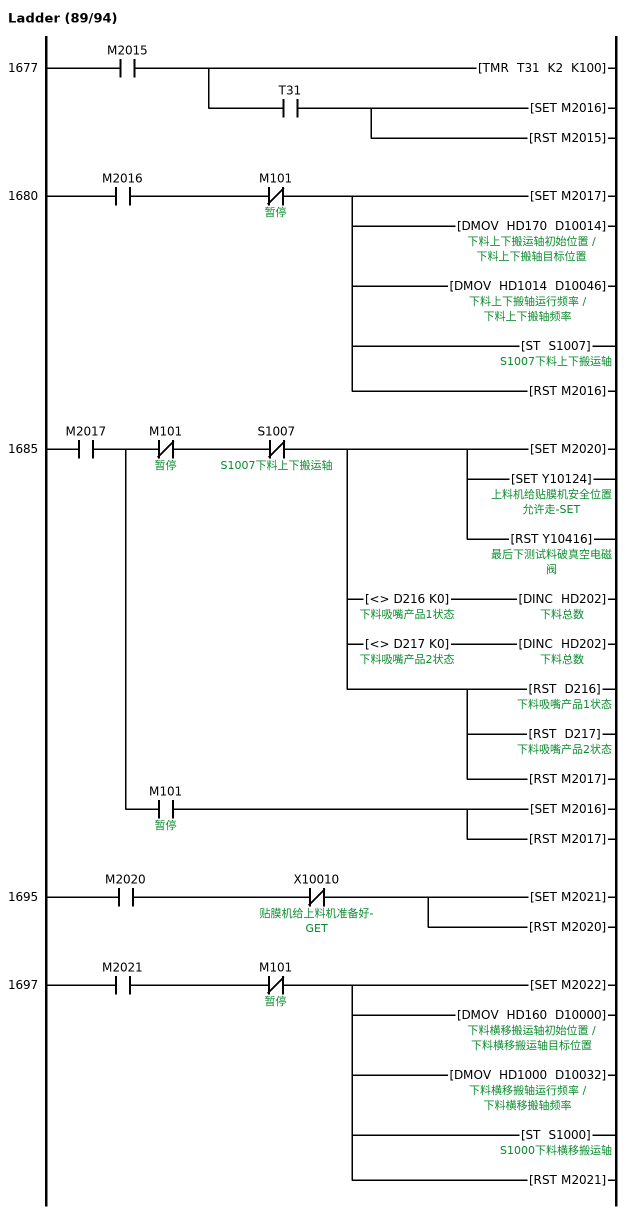
LD     M2015
TMR    T31 K2 K100
AND    T31
SET    M2016
RST    M2015
LD     M2016
ANI    M101	; 暂停
SET    M2017
DMOV   HD170 D10014	; 下料上下搬运轴初始位置 / 下料上下搬轴目标位置
DMOV   HD1014 D10046	; 下料上下搬轴运行频率 / 下料上下搬轴频率
ST     S1007	; S1007下料上下搬运轴
RST    M2016
LD     M2017
MPS
ANI    M101	; 暂停
ANI    S1007	; S1007下料上下搬运轴
SET    M2020
SET    Y10124	; 上料机给贴膜机安全位置允许走-SET
RST    Y10416	; 最后下测试料破真空电磁阀
MPS
AND<>  D216 K0	; 下料吸嘴产品1状态
DINC   HD202	; 下料总数
MRD
AND<>  D217 K0	; 下料吸嘴产品2状态
DINC   HD202	; 下料总数
MPP
RST    D216	; 下料吸嘴产品1状态
RST    D217	; 下料吸嘴产品2状态
RST    M2017
MPP
AND    M101	; 暂停
SET    M2016
RST    M2017
LD     M2020
ANI    X10010	; 贴膜机给上料机准备好-GET
SET    M2021
RST    M2020
LD     M2021
ANI    M101	; 暂停
SET    M2022
DMOV   HD160 D10000	; 下料横移搬运轴初始位置 / 下料横移搬运轴目标位置
DMOV   HD1000 D10032	; 下料横移搬轴运行频率 / 下料横移搬轴频率
ST     S1000	; S1000下料横移搬运轴
RST    M2021

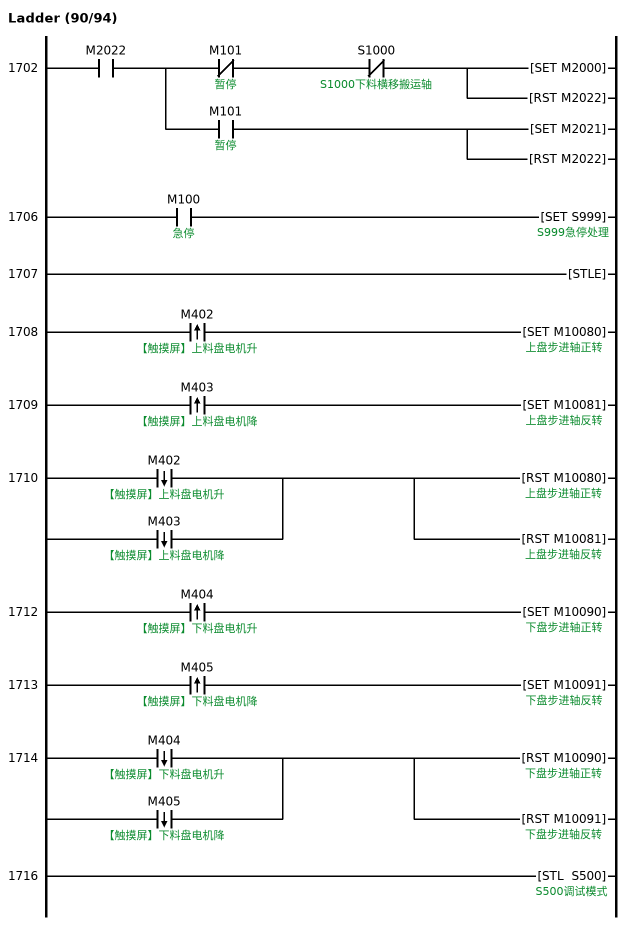
LD     M2022
MPS
ANI    M101	; 暂停
ANI    S1000	; S1000下料横移搬运轴
SET    M2000
RST    M2022
MPP
AND    M101	; 暂停
SET    M2021
RST    M2022
LD     M100	; 急停
SET    S999	; S999急停处理
STLE
LDP    M402	; 【触摸屏】上料盘电机升
SET    M10080	; 上盘步进轴正转
LDP    M403	; 【触摸屏】上料盘电机降
SET    M10081	; 上盘步进轴反转
LDF    M402	; 【触摸屏】上料盘电机升
ORF    M403	; 【触摸屏】上料盘电机降
RST    M10080	; 上盘步进轴正转
RST    M10081	; 上盘步进轴反转
LDP    M404	; 【触摸屏】下料盘电机升
SET    M10090	; 下盘步进轴正转
LDP    M405	; 【触摸屏】下料盘电机降
SET    M10091	; 下盘步进轴反转
LDF    M404	; 【触摸屏】下料盘电机升
ORF    M405	; 【触摸屏】下料盘电机降
RST    M10090	; 下盘步进轴正转
RST    M10091	; 下盘步进轴反转
STL    S500	; S500调试模式

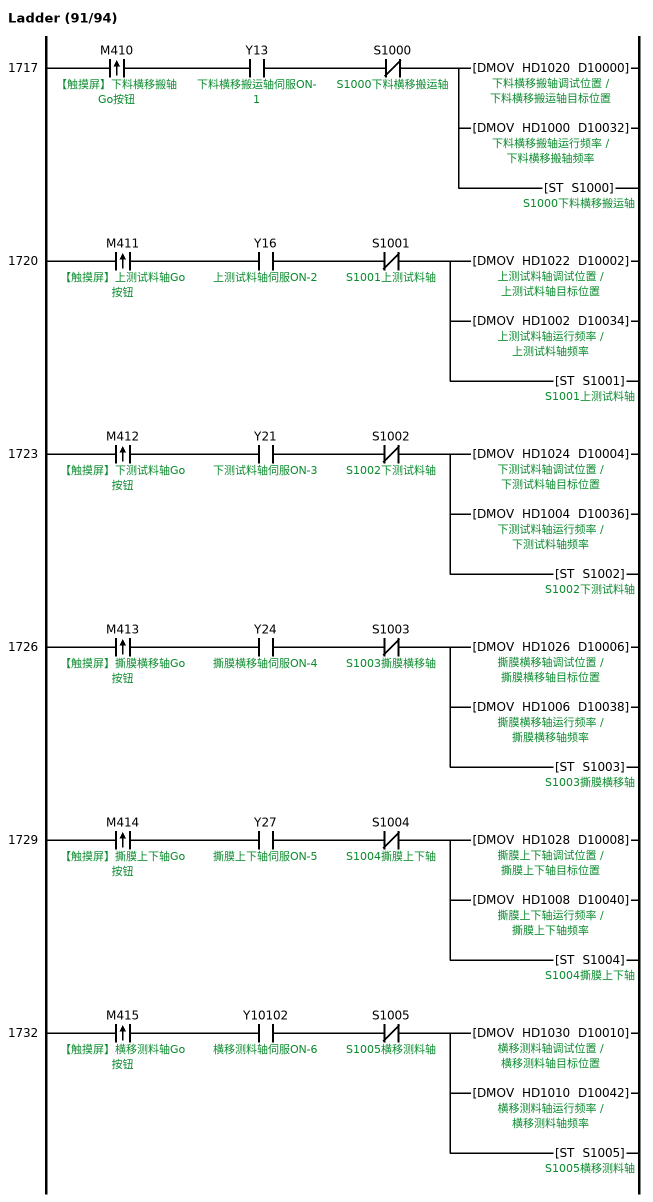
LDP    M410	; 【触摸屏】下料横移搬轴Go按钮
AND    Y13	; 下料横移搬运轴伺服ON-1
ANI    S1000	; S1000下料横移搬运轴
DMOV   HD1020 D10000	; 下料横移搬轴调试位置 / 下料横移搬运轴目标位置
DMOV   HD1000 D10032	; 下料横移搬轴运行频率 / 下料横移搬轴频率
ST     S1000	; S1000下料横移搬运轴
LDP    M411	; 【触摸屏】上测试料轴Go按钮
AND    Y16	; 上测试料轴伺服ON-2
ANI    S1001	; S1001上测试料轴
DMOV   HD1022 D10002	; 上测试料轴调试位置 / 上测试料轴目标位置
DMOV   HD1002 D10034	; 上测试料轴运行频率 / 上测试料轴频率
ST     S1001	; S1001上测试料轴
LDP    M412	; 【触摸屏】下测试料轴Go按钮
AND    Y21	; 下测试料轴伺服ON-3
ANI    S1002	; S1002下测试料轴
DMOV   HD1024 D10004	; 下测试料轴调试位置 / 下测试料轴目标位置
DMOV   HD1004 D10036	; 下测试料轴运行频率 / 下测试料轴频率
ST     S1002	; S1002下测试料轴
LDP    M413	; 【触摸屏】撕膜横移轴Go按钮
AND    Y24	; 撕膜横移轴伺服ON-4
ANI    S1003	; S1003撕膜横移轴
DMOV   HD1026 D10006	; 撕膜横移轴调试位置 / 撕膜横移轴目标位置
DMOV   HD1006 D10038	; 撕膜横移轴运行频率 / 撕膜横移轴频率
ST     S1003	; S1003撕膜横移轴
LDP    M414	; 【触摸屏】撕膜上下轴Go按钮
AND    Y27	; 撕膜上下轴伺服ON-5
ANI    S1004	; S1004撕膜上下轴
DMOV   HD1028 D10008	; 撕膜上下轴调试位置 / 撕膜上下轴目标位置
DMOV   HD1008 D10040	; 撕膜上下轴运行频率 / 撕膜上下轴频率
ST     S1004	; S1004撕膜上下轴
LDP    M415	; 【触摸屏】横移测料轴Go按钮
AND    Y10102	; 横移测料轴伺服ON-6
ANI    S1005	; S1005横移测料轴
DMOV   HD1030 D10010	; 横移测料轴调试位置 / 横移测料轴目标位置
DMOV   HD1010 D10042	; 横移测料轴运行频率 / 横移测料轴频率
ST     S1005	; S1005横移测料轴

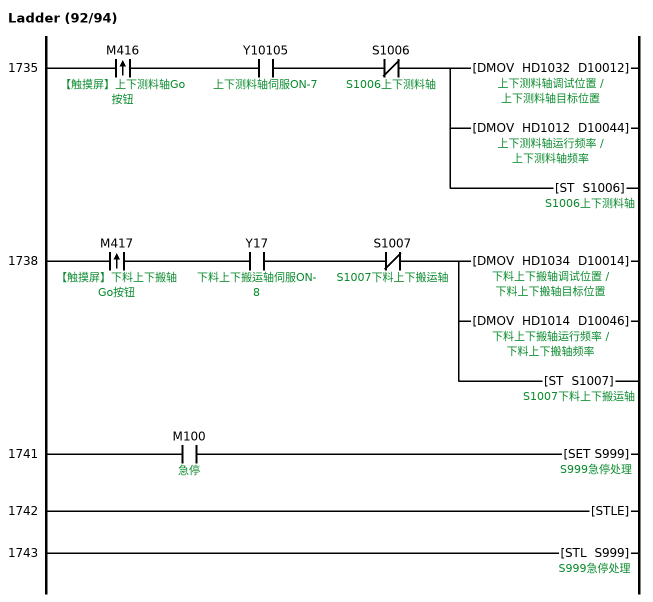
LDP    M416	; 【触摸屏】上下测料轴Go按钮
AND    Y10105	; 上下测料轴伺服ON-7
ANI    S1006	; S1006上下测料轴
DMOV   HD1032 D10012	; 上下测料轴调试位置 / 上下测料轴目标位置
DMOV   HD1012 D10044	; 上下测料轴运行频率 / 上下测料轴频率
ST     S1006	; S1006上下测料轴
LDP    M417	; 【触摸屏】下料上下搬轴Go按钮
AND    Y17	; 下料上下搬运轴伺服ON-8
ANI    S1007	; S1007下料上下搬运轴
DMOV   HD1034 D10014	; 下料上下搬轴调试位置 / 下料上下搬轴目标位置
DMOV   HD1014 D10046	; 下料上下搬轴运行频率 / 下料上下搬轴频率
ST     S1007	; S1007下料上下搬运轴
LD     M100	; 急停
SET    S999	; S999急停处理
STLE
STL    S999	; S999急停处理

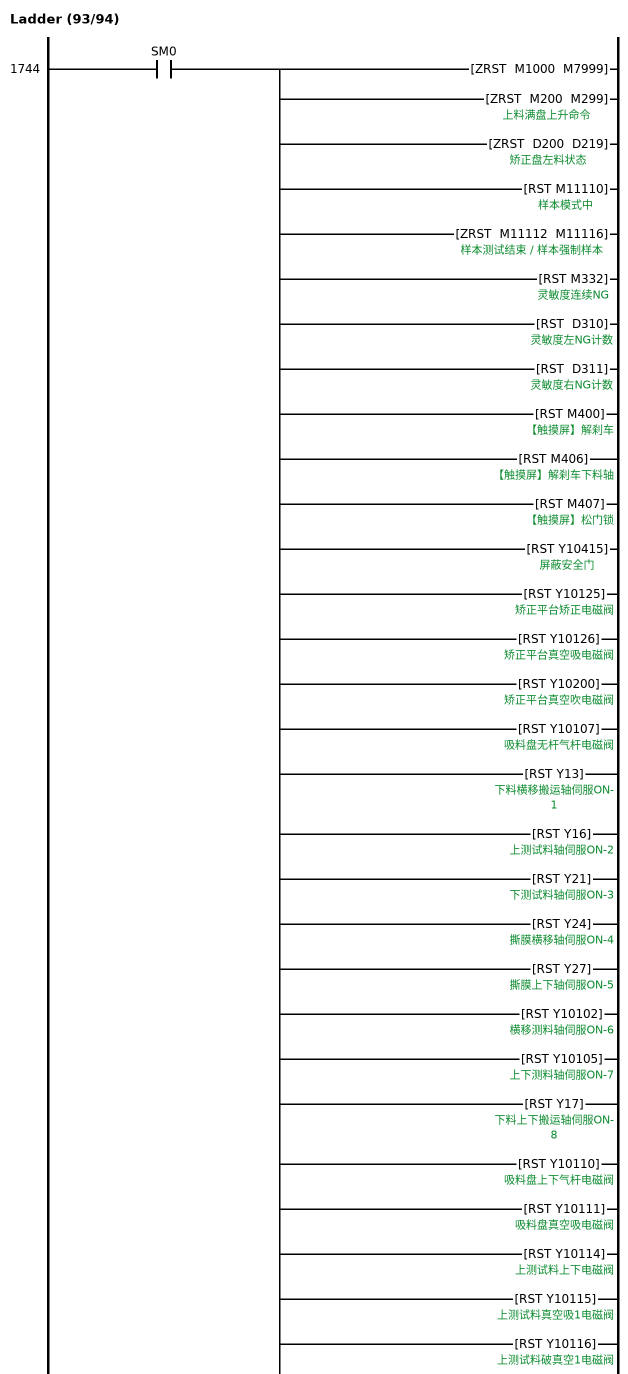
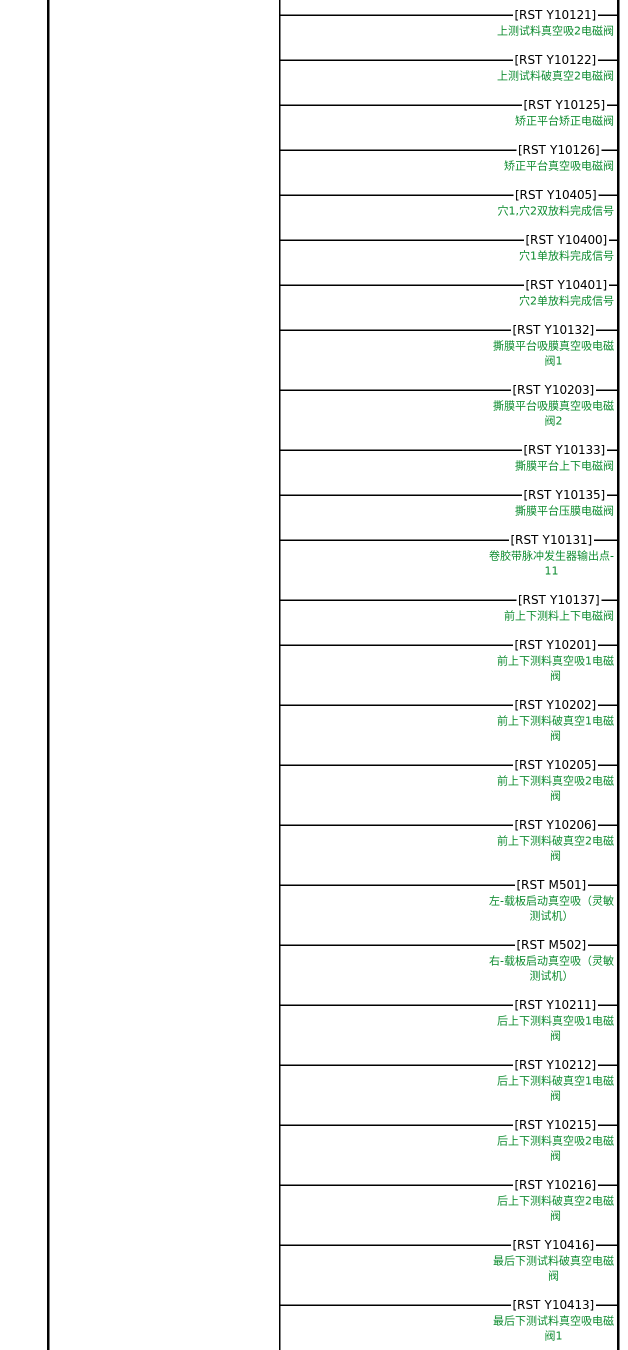
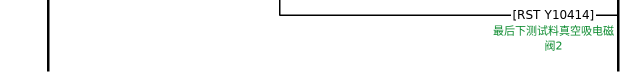
LD     SM0
ZRST   M1000 M7999
ZRST   M200 M299	; 上料满盘上升命令
ZRST   D200 D219	; 矫正盘左料状态
RST    M11110	; 样本模式中
ZRST   M11112 M11116	; 样本测试结束 / 样本强制样本
RST    M332	; 灵敏度连续NG
RST    D310	; 灵敏度左NG计数
RST    D311	; 灵敏度右NG计数
RST    M400	; 【触摸屏】解刹车
RST    M406	; 【触摸屏】解刹车下料轴
RST    M407	; 【触摸屏】松门锁
RST    Y10415	; 屏蔽安全门
RST    Y10125	; 矫正平台矫正电磁阀
RST    Y10126	; 矫正平台真空吸电磁阀
RST    Y10200	; 矫正平台真空吹电磁阀
RST    Y10107	; 吸料盘无杆气杆电磁阀
RST    Y13	; 下料横移搬运轴伺服ON-1
RST    Y16	; 上测试料轴伺服ON-2
RST    Y21	; 下测试料轴伺服ON-3
RST    Y24	; 撕膜横移轴伺服ON-4
RST    Y27	; 撕膜上下轴伺服ON-5
RST    Y10102	; 横移测料轴伺服ON-6
RST    Y10105	; 上下测料轴伺服ON-7
RST    Y17	; 下料上下搬运轴伺服ON-8
RST    Y10110	; 吸料盘上下气杆电磁阀
RST    Y10111	; 吸料盘真空吸电磁阀
RST    Y10114	; 上测试料上下电磁阀
RST    Y10115	; 上测试料真空吸1电磁阀
RST    Y10116	; 上测试料破真空1电磁阀
RST    Y10121	; 上测试料真空吸2电磁阀
RST    Y10122	; 上测试料破真空2电磁阀
RST    Y10125	; 矫正平台矫正电磁阀
RST    Y10126	; 矫正平台真空吸电磁阀
RST    Y10405	; 穴1,穴2双放料完成信号
RST    Y10400	; 穴1单放料完成信号
RST    Y10401	; 穴2单放料完成信号
RST    Y10132	; 撕膜平台吸膜真空吸电磁阀1
RST    Y10203	; 撕膜平台吸膜真空吸电磁阀2
RST    Y10133	; 撕膜平台上下电磁阀
RST    Y10135	; 撕膜平台压膜电磁阀
RST    Y10131	; 卷胶带脉冲发生器输出点-11
RST    Y10137	; 前上下测料上下电磁阀
RST    Y10201	; 前上下测料真空吸1电磁阀
RST    Y10202	; 前上下测料破真空1电磁阀
RST    Y10205	; 前上下测料真空吸2电磁阀
RST    Y10206	; 前上下测料破真空2电磁阀
RST    M501	; 左-载板启动真空吸（灵敏测试机）
RST    M502	; 右-载板启动真空吸（灵敏测试机）
RST    Y10211	; 后上下测料真空吸1电磁阀
RST    Y10212	; 后上下测料破真空1电磁阀
RST    Y10215	; 后上下测料真空吸2电磁阀
RST    Y10216	; 后上下测料破真空2电磁阀
RST    Y10416	; 最后下测试料破真空电磁阀
RST    Y10413	; 最后下测试料真空吸电磁阀1
RST    Y10414	; 最后下测试料真空吸电磁阀2

